FUNCTION TryConvert_BYTE_TO_BOOL : BOOL
VAR_INPUT
	in : BYTE;
	out : REFERENCE TO BOOL;
END_VAR

out := BYTE_TO_BOOL(in);
TryConvert_BYTE_TO_BOOL := TRUE;

END_FUNCTION

(* stored: Version 1.1.0.1, ProductVersion 3.1.4024.12
   POU TryConvert_BYTE_TO_BOOL: Id {4839c443-3dea-49ad-a6eb-5f2a029176cb}, SpecialFunc None *)
